(* IEC 61131-3 sources: programs/VI-54/VI-54_20171205/VI-54_20171205/Stations/PLC_VI54/VI-54_171014/Class/String, 1 file *)

(* ---- String.st ---- *)
(*!
<Class
	Name               = "String"
	Revision           = "1.10"
	RealtimeTask       = "false"
	CyclicTask         = "false"
	BackgroundTask     = "false"
	Sigmatek           = "true"
	OSInterface        = "false"
	HighPriority       = "false"
	Automatic          = "false"
	UpdateMode         = "Prescan"
	IconPath           = ".\Class\String\aString.ICO"
	SharedCommandTable = "true"
	Objectsize         = "(300,120)"
	Comment            = "handels character strings">
	<Channels>
		<Server
			Name           = "Data"
			Initialize     = "true"
			Visualized     = "true"
			WriteProtected = "false"
			Comment        = "use this channel to access the string functions">
		</Server>
		<Client Name="MerkerEx0" Required="true" Internal="true"/>
	</Channels>
	<RevDoku>
		<Owner Company="Sigmatek Gmbh &amp; Co KG"/>
		<Dokumentation Revision="1.10" Date="2012-11-05" Author="spimar" Company="Sigmatek Gmbh &amp; Co KG" Description="New client (SingleRealloc) which is used for an optimized memory handling!"/>
	</RevDoku>
	<Network Name="String">
		<!-- List of Components in this network -->
		<Components>
			<Object
				Name       = "_base"
				Class      = "StringInternal"
				Position   = "(720,360)"
				Visualized = "true">
				<Channels>
					<Server Name="Data"/>
					<Client Name="DataBuffer"/>
					<Client Name="SingleRealloc"/>
				</Channels>
			</Object>
			<Object
				Name       = "MerkerEx0"
				Class      = "MerkerEx"
				Position   = "(300,360)"
				Visualized = "true">
				<Channels>
					<Server Name="m_udLength"/>
					<Client Name="ThreadSafe" Value="0"/>
				</Channels>
			</Object>
		</Components>
		<Comments>
		</Comments>
		<!-- List of Connections in this network -->
		<Connections>
			<Connection Source="_base.DataBuffer" Destination="MerkerEx0.m_udLength" Vertices="(720,450),(736,450),"/>
			<Connection Source="this.Data" Destination="_base.Data" Vertices="(1192,210),(1020,450),"/>
			<Connection Source="this.MerkerEx0" Destination="MerkerEx0.m_udLength"/>
			<Connection Source="_base.SingleRealloc" Destination="this.SingleRealloc" Vertices="(720,510),(240,510),(240,210),(38,210),"/>
		</Connections>
		<!-- Headerfiles -->
		<Options>
		</Options>
	</Network>
</Class>
*)
#pragma using StringInternal

String : CLASS
: StringInternal
  //Servers:
  //Clients:
	MerkerEx0 	: CltChCmd_MerkerEx;
  //Variables:
  //Functions:
  //Tables:
	FUNCTION @STD
		VAR_OUTPUT
			ret_code	: CONFSTATES;
		END_VAR;
	FUNCTION GLOBAL TAB @CT_;
END_CLASS;

#pragma using MerkerEx
